// TIA Portal V19 export
FUNCTION_BLOCK "Main_Safety_RTG1"   // FB128, F_LAD
   VAR
      ACK_GL : ACK_GL;
      F_Estop : "F_Estop_FB";
      F_Bimanuals : "F_TwoHands_FB";
      F_Zone00 : "F_Zone00_FB";
      F_Zone01_02_03 : "F_Zone01_02_03_FB";
      F_Zone05 : "F_Zone05_FB";
      F_Zone10 : "F_Zone10_FB";
      F_Zone11 : "F_Zone11_FB";
      F_Zone13 : "F_Zone13_FB";
      F_Zone15 : "F_Zone15_FB";
      F_Zone20 : "F_Zone20_FB";
      F_Zone21 : "F_Zone21_FB";
      F_Zone23 : "F_Zone23_FB";
      F_Zone25 : "F_Zone25_FB";
      F_Zone27 : "F_Zone27_FB";
      F_Zone29 : "F_Zone29_FB";
   END_VAR
   VAR_TEMP
      NOT_USED : Bool;
   END_VAR
BEGIN

REGION Network 2: Cumulative safety reset
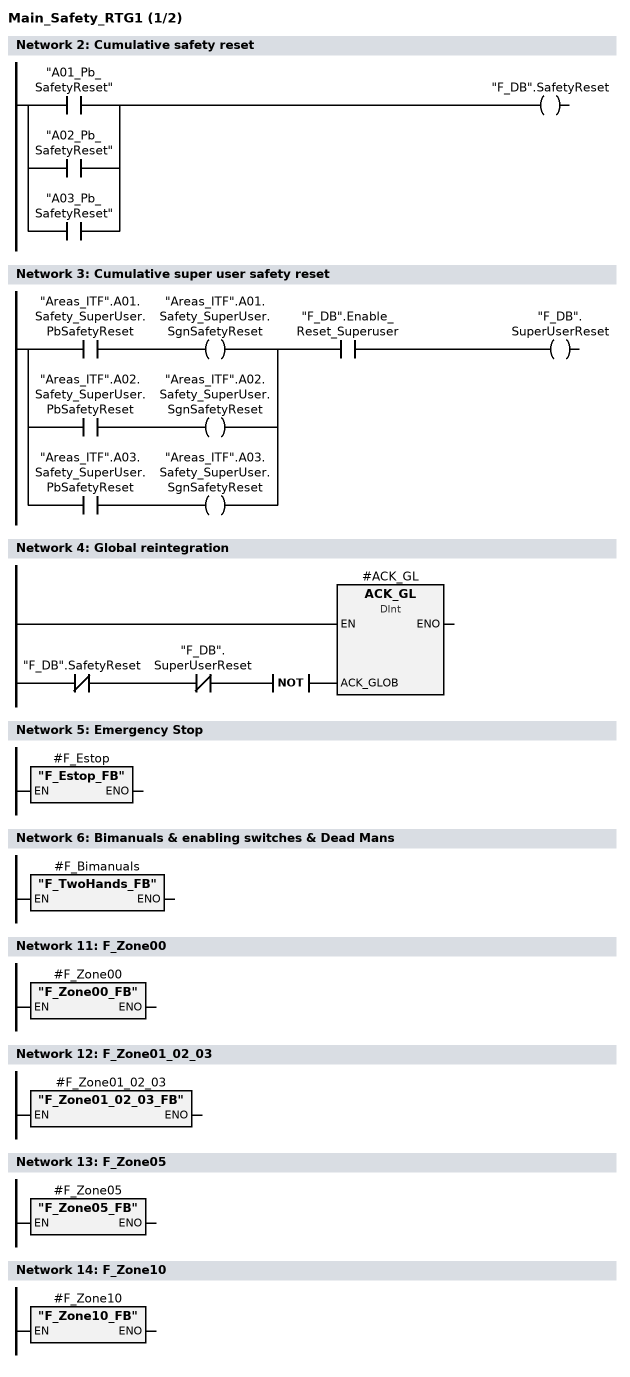
   RUNG wire#powerrail
      Contact( "A01_Pb_SafetyReset" )
      wire#w1
      Coil( "F_DB".SafetyReset )
   END_RUNG
   RUNG wire#powerrail
      Contact( "A02_Pb_SafetyReset" )
   END_RUNG wire#w1
   RUNG wire#powerrail
      Contact( "A03_Pb_SafetyReset" )
   END_RUNG wire#w1
   // the same network as SCL:
   "F_DB".SafetyReset := "A01_Pb_SafetyReset" OR "A02_Pb_SafetyReset" OR "A03_Pb_SafetyReset";
END_REGION

REGION Network 3: Cumulative super user safety reset
   RUNG wire#powerrail
      Contact( "Areas_ITF".A01.Safety_SuperUser.PbSafetyReset )
      Coil( "Areas_ITF".A01.Safety_SuperUser.SgnSafetyReset )
      wire#w1
      Contact( "F_DB".Enable_Reset_Superuser )
      Coil( "F_DB".SuperUserReset )
   END_RUNG
   RUNG wire#powerrail
      Contact( "Areas_ITF".A02.Safety_SuperUser.PbSafetyReset )
      Coil( "Areas_ITF".A02.Safety_SuperUser.SgnSafetyReset )
   END_RUNG wire#w1
   RUNG wire#powerrail
      Contact( "Areas_ITF".A03.Safety_SuperUser.PbSafetyReset )
      Coil( "Areas_ITF".A03.Safety_SuperUser.SgnSafetyReset )
   END_RUNG wire#w1
   // the same network as SCL:
   "Areas_ITF".A01.Safety_SuperUser.SgnSafetyReset := "Areas_ITF".A01.Safety_SuperUser.PbSafetyReset;
   "Areas_ITF".A02.Safety_SuperUser.SgnSafetyReset := "Areas_ITF".A02.Safety_SuperUser.PbSafetyReset;
   "Areas_ITF".A03.Safety_SuperUser.SgnSafetyReset := "Areas_ITF".A03.Safety_SuperUser.PbSafetyReset;
   "F_DB".SuperUserReset := ("Areas_ITF".A01.Safety_SuperUser.PbSafetyReset OR "Areas_ITF".A02.Safety_SuperUser.PbSafetyReset OR "Areas_ITF".A03.Safety_SuperUser.PbSafetyReset) AND "F_DB".Enable_Reset_Superuser;
END_REGION

REGION Network 4: Global reintegration
   RUNG wire#powerrail
      { S7_Templates := "codedbool_type := DInt" } #ACK_GL.ACK_GL(ACK_GLOB := wire#w1)
   END_RUNG
   RUNG wire#powerrail
      I_Contact( "F_DB".SafetyReset )
      I_Contact( "F_DB".SuperUserReset )
      Not()
   END_RUNG wire#w1
   // the same network as SCL:
   #ACK_GL(ACK_GLOB := NOT (NOT "F_DB".SafetyReset AND NOT "F_DB".SuperUserReset));   // ACK_GL
END_REGION

REGION Network 5: Emergency Stop
   RUNG wire#powerrail
      #F_Estop()
   END_RUNG
   // the same network as SCL:
   #F_Estop();   // "F_Estop_FB"
END_REGION

REGION Network 6: Bimanuals & enabling switches & Dead Mans
   RUNG wire#powerrail
      #F_Bimanuals()
   END_RUNG
   // the same network as SCL:
   #F_Bimanuals();   // "F_TwoHands_FB"
END_REGION

REGION Network 7: >
END_REGION

REGION Network 8: >
END_REGION

REGION Network 9: >
END_REGION

REGION Network 10: ######################### SAFETY ZONES OF AREA 01 #########################
END_REGION

REGION Network 11: F_Zone00
   RUNG wire#powerrail
      #F_Zone00()
   END_RUNG
   // the same network as SCL:
   #F_Zone00();   // "F_Zone00_FB"
END_REGION

REGION Network 12: F_Zone01_02_03
   RUNG wire#powerrail
      #F_Zone01_02_03()
   END_RUNG
   // the same network as SCL:
   #F_Zone01_02_03();   // "F_Zone01_02_03_FB"
END_REGION

REGION Network 13: F_Zone05
   RUNG wire#powerrail
      #F_Zone05()
   END_RUNG
   // the same network as SCL:
   #F_Zone05();   // "F_Zone05_FB"
END_REGION

REGION Network 14: F_Zone10
   RUNG wire#powerrail
      #F_Zone10()
   END_RUNG
   // the same network as SCL:
   #F_Zone10();   // "F_Zone10_FB"
END_REGION

REGION Network 15: >
END_REGION

REGION Network 16: >
END_REGION

REGION Network 17: ######################### SAFETY ZONES OF AREA 02 #########################
END_REGION

REGION Network 18: F Zone 11
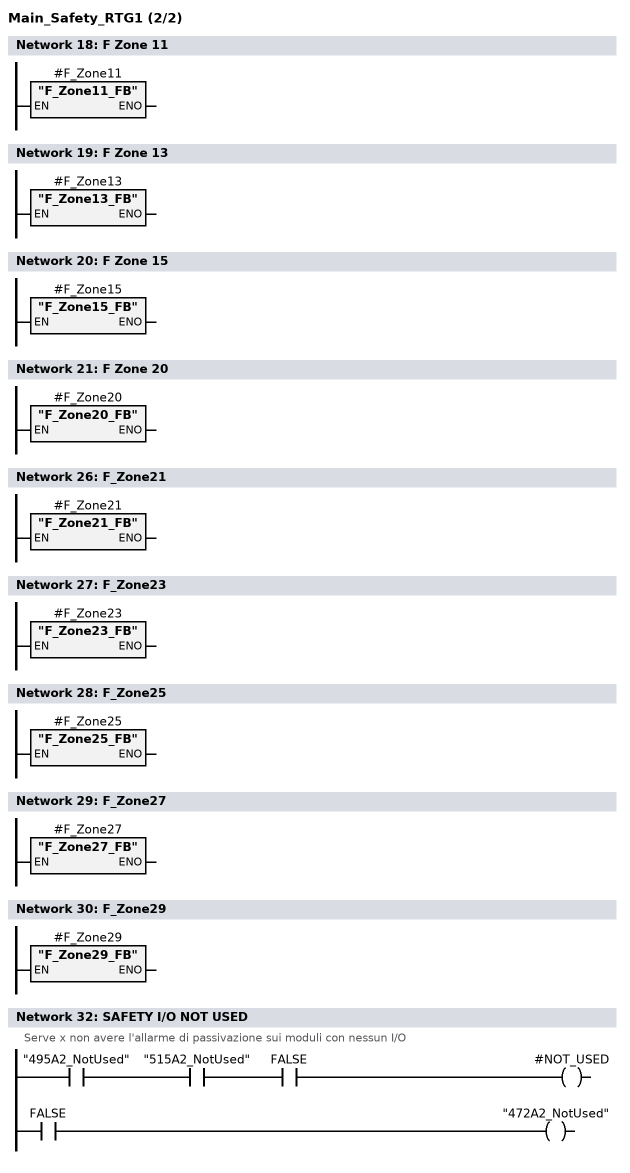
   RUNG wire#powerrail
      #F_Zone11()
   END_RUNG
   // the same network as SCL:
   #F_Zone11();   // "F_Zone11_FB"
END_REGION

REGION Network 19: F Zone 13
   RUNG wire#powerrail
      #F_Zone13()
   END_RUNG
   // the same network as SCL:
   #F_Zone13();   // "F_Zone13_FB"
END_REGION

REGION Network 20: F Zone 15
   RUNG wire#powerrail
      #F_Zone15()
   END_RUNG
   // the same network as SCL:
   #F_Zone15();   // "F_Zone15_FB"
END_REGION

REGION Network 21: F Zone 20
   RUNG wire#powerrail
      #F_Zone20()
   END_RUNG
   // the same network as SCL:
   #F_Zone20();   // "F_Zone20_FB"
END_REGION

REGION Network 22: >
END_REGION

REGION Network 23: >
END_REGION

REGION Network 24: >
END_REGION

REGION Network 25: ######################### SAFETY ZONES OF AREA 03 #########################
END_REGION

REGION Network 26: F_Zone21
   RUNG wire#powerrail
      #F_Zone21()
   END_RUNG
   // the same network as SCL:
   #F_Zone21();   // "F_Zone21_FB"
END_REGION

REGION Network 27: F_Zone23
   RUNG wire#powerrail
      #F_Zone23()
   END_RUNG
   // the same network as SCL:
   #F_Zone23();   // "F_Zone23_FB"
END_REGION

REGION Network 28: F_Zone25
   RUNG wire#powerrail
      #F_Zone25()
   END_RUNG
   // the same network as SCL:
   #F_Zone25();   // "F_Zone25_FB"
END_REGION

REGION Network 29: F_Zone27
   RUNG wire#powerrail
      #F_Zone27()
   END_RUNG
   // the same network as SCL:
   #F_Zone27();   // "F_Zone27_FB"
END_REGION

REGION Network 30: F_Zone29
   RUNG wire#powerrail
      #F_Zone29()
   END_RUNG
   // the same network as SCL:
   #F_Zone29();   // "F_Zone29_FB"
END_REGION

REGION Network 31: >
END_REGION

REGION Network 32: SAFETY I/O NOT USED
   // Serve x non avere l'allarme di passivazione sui moduli con nessun I/O
   RUNG wire#powerrail
      Contact( "495A2_NotUsed" )
      Contact( "515A2_NotUsed" )
      Contact( FALSE )
      Coil( #NOT_USED )
   END_RUNG
   RUNG wire#powerrail
      Contact( FALSE )
      Coil( "472A2_NotUsed" )
   END_RUNG
   // the same network as SCL:
   #NOT_USED := "495A2_NotUsed" AND "515A2_NotUsed" AND FALSE;
   "472A2_NotUsed" := FALSE;
END_REGION

REGION Network 33: NOT USED OUTPUT
END_REGION

REGION Network 34: >
END_REGION

REGION Network 35: >
END_REGION
END_FUNCTION_BLOCK
